(* Logix 5000 project; controller axis1 vendor 1 type 14 code 155 rev 20.12; software revision 20.01 *)

TASK MainTask (continuous, watchdog 500 ms) : MainProgram

MODULES
   Local : vendor 1 type 14 code 155 (PointIO 0, rev 20.12)
      Kinetix_350 : vendor 1 type 37 code 27 (Ethernet 192.168.1.7, rev 1.1, MotionDiagnostics RPI 1 ms, MotionSync RPI 2 ms)
      XG_7702 : ETHERNET-MODULE (Ethernet 192.168.1.6, rev 1.1, Output RPI 10 ms)
       : 1734-IE2V (PointIO 2, rev 3.1, Input RPI 80 ms)
       : vendor 10 type 150 code 185 (PointIO 5, rev 1.1, Output RPI 50 ms)
      Discrete_IO : Embedded (PointIO 1, rev 20.11, Output RPI 20 ms)
       : 1734-OE2V (PointIO 3, rev 3.1, Output RPI 80 ms)
       : vendor 1 type 109 code 13 (PointIO 4, rev 3.1, Output RPI 80 ms)
END_MODULES

VAR_GLOBAL   (* controller tags *)
   Axis_1 : AXIS_CIP_DRIVE;
   Kinetix_350_Quick_Start : MOTION_GROUP;
END_VAR

PROGRAM MainProgram   (* main routine MainRoutine *)
VAR
   Axis1_Motion : MOTION_INSTRUCTION;
   light : BOOL := 1;
   Move_Incr_Axis_1 : MOTION_INSTRUCTION;
   one_shot1 : BOOL;
   start : BOOL;
   Timer1 : TIMER := (PRE := 50);
   Timer2 : TIMER := (PRE := 50);
END_VAR

ROUTINE MainRoutine   (* ladder *)
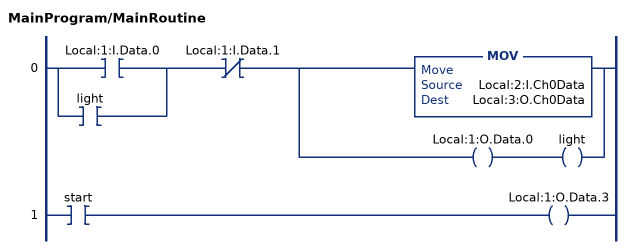
   0: [XIC(Local:1:I.Data.0) ,XIC(light) ]XIO(Local:1:I.Data.1)[MOV(Local:2:I.Ch0Data,Local:3:O.Ch0Data) ,OTE(Local:1:O.Data.0) OTE(light) ];
   1: XIC(start)OTE(Local:1:O.Data.3);
END_ROUTINE
END_PROGRAM
